    _moveParam.Axis1.Position := _multiAxis.Axis_1.AxisStatus.ActPos + 10000;
    _moveParam.Axis1.Velocity := _velocity;
    _moveParam.Axis1.Acceleration := _acceleration;
    _moveParam.Axis1.Deceleration := _deceleration;
    _moveParam.Axis1.Jerk := _jerk;
    _moveParam.Axis2.Position := _multiAxis.Axis_2.AxisStatus.ActPos - 1000;
    _moveParam.Axis2.Velocity := _velocity;
    _moveParam.Axis2.Acceleration := _acceleration;
    _moveParam.Axis2.Deceleration := _deceleration;
    _moveParam.Axis2.Jerk := _jerk;
    _moveParam.Axis3.Position := _multiAxis.Axis_3.AxisStatus.ActPos - 1000;
    _moveParam.Axis3.Velocity := _velocity;
    _moveParam.Axis3.Acceleration := _acceleration;
    _moveParam.Axis3.Deceleration := _deceleration;
    _moveParam.Axis3.Jerk := _jerk;
    _moveParam.Axis4.Position := _multiAxis.Axis_4.AxisStatus.ActPos - 1000;
    _moveParam.Axis4.Velocity := _velocity;
    _moveParam.Axis4.Acceleration := _acceleration;
    _moveParam.Axis4.Deceleration := _deceleration;
    _moveParam.Axis4.Jerk := _jerk;

    IF _multiAxis.MoveAbsolute(_moveParam).Done THEN
        seq.CompleteStep();
    END_IF
    //--------------------------------------------------------
END_IF;

IF (seq.Step(inStepID := 600, inEnabled := TRUE, inStepDescription := 'ASKING FOR RESTORING')) THEN
    //--------------------------------------------------------
    answer := _dialog.Show()
        .WithType(eDialogType.Question)
        .WithCaption('Question?')
        .WithText('Do you want to restore MultiAxis component?')
        .WithYesNo().Answer;

    //
    IF (answer = TcoCore.eDialogAnswer.Yes) THEN
        _multiAxis.Restore();
        seq.CompleteStep();
    ELSIF (answer = TcoCore.eDialogAnswer.No) THEN
        _sequence1Task.Restore();
    END_IF;
    //--------------------------------------------------------
END_IF;

IF (seq.Step(inStepID := seq.RESTORE_STEP_ID, inEnabled := TRUE, inStepDescription := 'RETURN TO THE START OF THE SEQUENCE')) THEN
    //--------------------------------------------------------
    seq.CompleteSequence();
    //--------------------------------------------------------
END_IF;

seq.Close();
END_METHOD

END_FUNCTION_BLOCK

// ---- Tests/TcoContext/WrappedComponent/WrappedComponentExample.TcPOU
FUNCTION_BLOCK WrappedComponentExample EXTENDS TcoCore.TcoComponent
VAR_OUTPUT
END_VAR
VAR
    _config : WrappedComponentExample_Config;
    _status : WrappedComponentExample_Status;
    _control : WrappedComponentExample_Control;
    _components : WrappedComponentsExample := (Parent := THIS^);
    _throwTask : TcoCore.TcoTask(THIS^);
    _restoreTask : TcoCore.TcoTask(THIS^);
END_VAR

PROPERTY Components : REFERENCE TO WrappedComponentsExample
GET
Components ref= _components;
END_GET
END_PROPERTY

(*~
    <docu>
        <summary>
            Restores this instance to the Ready state. Can be called explicitly or from within one of the restore mechanisms.
        </summary>
    </docu>
~*)
METHOD Restore : ITcoRestorable
END_METHOD

(*~
    <docu>
        <summary>
            Custom service (manual, maintenance) logic.
            This method must be implemented in derived class.
        </summary>
    </docu>
~*)
METHOD PROTECTED ServiceMode
END_METHOD

END_FUNCTION_BLOCK

// ---- Tests/TcoContext/Sequence1Task.TcPOU
FUNCTION_BLOCK Sequence1Task EXTENDS TcoCore.TcoTask
VAR_INPUT
    Sequence : TcoCore.ITcoSequencer;
END_VAR

(*~
    <docu>
        <summary>
            Restores this instance to the Ready state. Can be called explicitly or from within one of the restore mechanisms.
            <para>
                See also <see cref="PlcDocu.TcoCore.TcoTask.AutoRestorable()"/>
            </para>
        </summary>
    </docu>
~*)
METHOD Restore : ITcoRestorable
SUPER^.Restore();
THIS^.Sequence.Restore();
END_METHOD

END_FUNCTION_BLOCK
